Universal Robots PolyScope program: partmover05_amp.urp

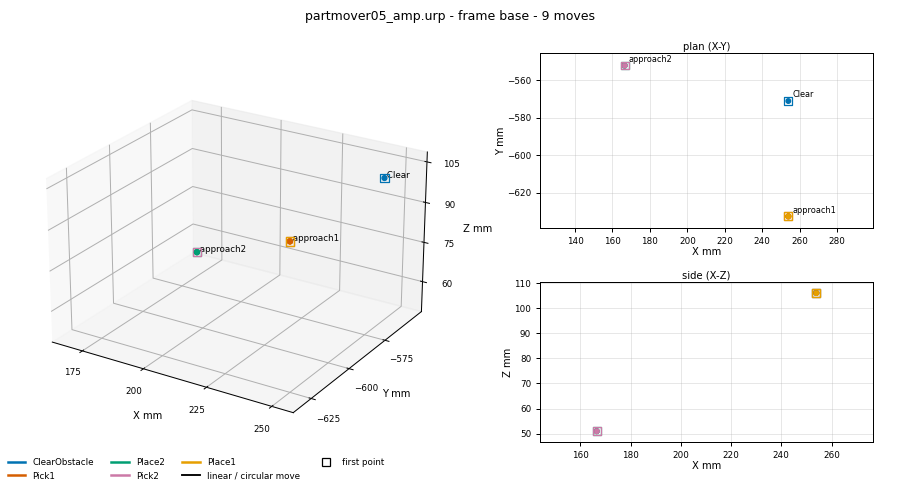
[picture p0: tool path of partmover05_amp.urp in frame base, 9 of 9 moves have a stored position in this frame; points joined in program order, loops and branches not executed]
Program partmover05_amp (installation=default directory=/programs createdIn=5.9.1.1031110 lastSavedIn=5.9.1.1031110 robotSerialNumber=20195501059)
Calibrated DH parameters: a=[0.000146, -0.418764, -0.053981, 0.000058, -0.000023, 0]; d=[0.162545, 37.319448, -206.067439, 168.881546, 0.09955, 0.099464]; alpha=[1.57004, -0.001979, 0.002304, 1.570607, -1.57066, 0]; deltaTheta=[0, -0.174616, -1.258233, 1.432844, -0.000001, 0]
InitVariablesNode
BeforeStart
  URCap Gripper Activate (Robotiq_Grippers, Robotiq Inc.) dataModel(ResetAndActivateKey=false)
  URCap Gripper (Robotiq_Grippers, Robotiq Inc.) dataModel(position=50.0, force=100.0, speed=100.0, positionInDouble=50.0, forceInDouble=100.0, speedInDouble=100.0, slaveIds=[9], blocking=true)
  Call ClearObstacle
Robot Program (runOnlyOnce=false)
  Call Pick1
  URCap Grip Check (Robotiq_Grippers, Robotiq Inc.) dataModel(ObjectDetectedKey=true, DimensionValidationKey=false, DimensionKey=100.0, DimensionDimensionPositiveGapKey=5.0, DimensionNegativeGapKey=5.0, GripperIdKey=1, ModelDefinedKey=true); state(isChildrenLocked=true)
    URCap If (Robotiq_Grippers, Robotiq Inc.)
      Call ClearObstacle
      Call Place2
  Call Pick2
  URCap Grip Check (Robotiq_Grippers, Robotiq Inc.) dataModel(ObjectDetectedKey=true, DimensionValidationKey=false, DimensionKey=100.0, DimensionDimensionPositiveGapKey=5.0, DimensionNegativeGapKey=5.0, GripperIdKey=1, ModelDefinedKey=true); state(isChildrenLocked=true)
    URCap If (Robotiq_Grippers, Robotiq Inc.)
      Call ClearObstacle
      Call Place1
SubProgram -> ClearObstacle
SubProgram -> Pick1
SubProgram -> Place2
SubProgram -> Pick2
SubProgram -> Place1
SubProgram ClearObstacle (keepSynchronizedWithDisk=false)
  MoveL speed 250 mm/s, acceleration 1200 mm/s^2 (useActiveTCP=true) feature=Base
    Waypoint Clear: TCP in base x=253.918 y=-571.009 z=106.037 mm, rx=-2.2358 ry=-2.207 rz=0 rad; joints [101.61, -67.822, 94.579, -116.748, 270.007, 102.367] deg; TCP offset x=0 y=0 z=174 mm, rx=0 ry=0 rz=0 rad
SubProgram Pick1 (keepSynchronizedWithDisk=false)
  MoveL speed 250 mm/s, acceleration 1200 mm/s^2 (useActiveTCP=true) feature=Base
    Waypoint approach1: TCP in base x=253.939 y=-632.617 z=106.042 mm, rx=2.2358 ry=2.207 rz=0 rad; joints [100.55, -60.732, 83.822, -113.083, 269.987, 101.297] deg
    URCap Gripper (Robotiq_Grippers, Robotiq Inc.) dataModel(position=100.0, force=100.0, speed=100.0, positionInDouble=100.0, forceInDouble=100.0, speedInDouble=100.0, slaveIds=[9], blocking=true)
    MoveDirectionNode (selectedDirection=ZPlus toolParams=0.02, 0.5) feature=Joint_6_name
      Until TOOL_CONTACT_DETECTION (allowActions=true retraction=0.003 decelerationAcceleration=1 decelerationAngularAcceleration=34.906585)
        URCap Gripper (Robotiq_Grippers, Robotiq Inc.) dataModel(position=50.0, force=100.0, speed=100.0, positionInDouble=50.0, forceInDouble=100.0, speedInDouble=100.0, slaveIds=[9], blocking=true)
        MoveDirectionNode (selectedDirection=ZPlus) feature=Joint_6_name
          Until DISTANCE (allowActions=false deceleration=3 distanceNodeType=STOP) Distance=0.015; motionParameters(blendRadius=0)
        URCap Gripper (Robotiq_Grippers, Robotiq Inc.) dataModel(position=100.0, force=100.0, speed=100.0, positionInDouble=100.0, forceInDouble=100.0, speedInDouble=100.0, slaveIds=[9], blocking=true)
      Until DISTANCE (allowActions=false deceleration=3 distanceNodeType=STOP) Distance=0.025; motionParameters(blendRadius=0)
    Waypoint approach1: TCP in base x=253.939 y=-632.617 z=106.042 mm, rx=2.2358 ry=2.207 rz=0 rad; joints [100.55, -60.732, 83.822, -113.083, 269.987, 101.297] deg
SubProgram Place2 (keepSynchronizedWithDisk=false)
  MoveL speed 250 mm/s, acceleration 1200 mm/s^2 (useActiveTCP=true) feature=Base
    Waypoint approach2: TCP in base x=166.497 y=-552.051 z=50.992 mm, rx=3.1415 ry=-0.0034 rz=0 rad; joints [93.363, -69.603, 106.655, -127.047, 270.03, 183.517] deg
    MoveDirectionNode (selectedDirection=ZPlus toolParams=0.02, 0.5) feature=Joint_6_name
      Until TOOL_CONTACT_DETECTION (allowActions=false retraction=0.001 decelerationAcceleration=1 decelerationAngularAcceleration=34.906585)
    URCap Gripper (Robotiq_Grippers, Robotiq Inc.) dataModel(position=49.80392156862745, force=100.0, speed=100.0, positionInDouble=49.80392156862745, forceInDouble=100.0, speedInDouble=100.0, slaveIds=[9], blocking=true)
    Waypoint approach2: TCP in base x=166.497 y=-552.051 z=50.992 mm, rx=3.1415 ry=-0.0034 rz=0 rad; joints [93.363, -69.603, 106.655, -127.047, 270.03, 183.517] deg
SubProgram Pick2 (keepSynchronizedWithDisk=false)
  MoveL speed 250 mm/s, acceleration 1200 mm/s^2 (useActiveTCP=true) feature=Base
    Waypoint approach2: TCP in base x=166.497 y=-552.051 z=50.992 mm, rx=3.1415 ry=-0.0034 rz=0 rad; joints [93.363, -69.603, 106.655, -127.047, 270.03, 183.517] deg
    URCap Gripper (Robotiq_Grippers, Robotiq Inc.) dataModel(position=100.0, force=100.0, speed=100.0, positionInDouble=100.0, forceInDouble=100.0, speedInDouble=100.0, slaveIds=[9], blocking=true)
    MoveDirectionNode (selectedDirection=ZPlus toolParams=0.02, 0.5) feature=Joint_6_name
      Until TOOL_CONTACT_DETECTION (allowActions=true retraction=0.003 decelerationAcceleration=1 decelerationAngularAcceleration=34.906585)
        URCap Gripper (Robotiq_Grippers, Robotiq Inc.) dataModel(position=49.80392156862745, force=100.0, speed=100.0, positionInDouble=49.80392156862745, forceInDouble=100.0, speedInDouble=100.0, slaveIds=[9], blocking=true)
        MoveDirectionNode (selectedDirection=ZPlus) feature=Joint_6_name
          Until DISTANCE (allowActions=false deceleration=3 distanceNodeType=STOP) Distance=0.015; motionParameters(blendRadius=0)
        URCap Gripper (Robotiq_Grippers, Robotiq Inc.) dataModel(position=100.0, force=100.0, speed=100.0, positionInDouble=100.0, forceInDouble=100.0, speedInDouble=100.0, slaveIds=[9], blocking=true)
      Until DISTANCE (allowActions=false deceleration=3 distanceNodeType=STOP) Distance=0.025; motionParameters(blendRadius=0)
    Waypoint approach2: TCP in base x=166.497 y=-552.051 z=50.992 mm, rx=3.1415 ry=-0.0034 rz=0 rad; joints [93.363, -69.603, 106.655, -127.047, 270.03, 183.517] deg
SubProgram Place1 (keepSynchronizedWithDisk=false)
  MoveL speed 250 mm/s, acceleration 1200 mm/s^2 (useActiveTCP=true) feature=Base
    Waypoint approach1: TCP in base x=253.939 y=-632.617 z=106.042 mm, rx=2.2358 ry=2.207 rz=0 rad; joints [100.55, -60.732, 83.822, -113.083, 269.987, 101.297] deg
    MoveDirectionNode (selectedDirection=ZPlus toolParams=0.02, 0.5) feature=Joint_6_name
      Until TOOL_CONTACT_DETECTION (allowActions=false retraction=0.001 decelerationAcceleration=1 decelerationAngularAcceleration=34.906585)
    URCap Gripper (Robotiq_Grippers, Robotiq Inc.) dataModel(position=49.80392156862745, force=100.0, speed=100.0, positionInDouble=49.80392156862745, forceInDouble=100.0, speedInDouble=100.0, slaveIds=[9], blocking=true)
    Waypoint approach1: TCP in base x=253.939 y=-632.617 z=106.042 mm, rx=2.2358 ry=2.207 rz=0 rad; joints [100.55, -60.732, 83.822, -113.083, 269.987, 101.297] deg
